// TwinCAT 3 PLC project Virtual_PLC
// ProgramVersion: 3.1.4024.0
// libraries:
//   Tc2_Standard, * (Beckhoff Automation GmbH)
//   Tc2_System, * (Beckhoff Automation GmbH)
//   Tc3_Module, * (Beckhoff Automation GmbH)
// project tree:
//   DUTs/ KlantToestand.TcDUT, KleurmachineToestand.TcDUT, MedewerkerToestand.TcDUT, schudmachineToestand.TcDUT
//   / GlobalTextList.TcGTLO, PlcTask.TcTTO, Visualization Manager.TcVMO (not stored), Visualization.TcVIS
//   GVLs/ GVL.TcGVL
//   POUs/ kleurmachine.TcPOU, Medewerker.TcPOU, Klant.TcPOU, schudmachine.TcPOU
//   VISUs/ Visu_main.TcVIS
// real-time tasks:
//   TASK PlcTask: cycle T#10ms, priority 20, ADS port 350

CONFIGURATION Virtual_PLC
    RESOURCE PLC ON TwinCAT3
        TASK PlcTask(INTERVAL := T#10ms, PRIORITY := 20);
        PROGRAM Medewerker WITH PlcTask : Medewerker;
        PROGRAM schudmachine WITH PlcTask : schudmachine;
        PROGRAM kleurmachine WITH PlcTask : kleurmachine;
        PROGRAM Klant WITH PlcTask : Klant;
    END_RESOURCE
END_CONFIGURATION

// ---- DUTs/KlantToestand.TcDUT
{attribute 'qualified_only'}
{attribute 'strict'}
TYPE KlantToestand :
(
	voorBalie := 0,
	wordtGeholpen,
	aanHetWachten,
	heeftVerf
);
END_TYPE

// ---- DUTs/KleurmachineToestand.TcDUT
{attribute 'qualified_only'}
{attribute 'strict'}
TYPE KleurmachineToestand :
(
	startup := 0,
	home,
	info,
	scan,
	wachtOpBlik,
	kleurToevoegen,
	klaarMetToevoegen
);
END_TYPE

// ---- DUTs/MedewerkerToestand.TcDUT
{attribute 'qualified_only'}
{attribute 'strict'}
TYPE MedewerkerToestand :
(
	wachtenOpKlant := 0,
	klantHelpen,
	verfMengen,
	verfGeven
);
END_TYPE

// ---- DUTs/schudmachineToestand.TcDUT
{attribute 'qualified_only'}
{attribute 'strict'}
TYPE schudmachineToestand :
(
	startup := 0,
	automode,
	blikKlemmen,
	blikSchudden
);
END_TYPE

// ---- GVLs/GVL.TcGVL
{attribute 'qualified_only'}
VAR_GLOBAL
	// Keuzes van de klant
	typeVerf 	: STRING := 'null';
	merkVerf 	: STRING := 'null';
	kleurVerf	: STRING := 'null';
	hoeveelVerf : STRING := 'null';
	
	// Opdracht voor kleurmachine
	verfOrder 	: ARRAY[1..4] OF STRING;
	
	// knoppen/sensoren kleurmachine
	homeKnop : BOOL;
	okeKnop : BOOL;
	blikPresent : BOOL;
	opdrachtKnop : BOOL;
	startKnop : BOOL;	
	
	barcodeBlik : INT;
	
	// klant variabelen
	klantWiltVerf : BOOL := TRUE;
	klantWordtGeholpen : BOOL;
	klantWacht : BOOL;
	verfAanKlantGegeven : BOOL;
	
	// schudmachine variabelen
	schudmachineReady : BOOL := FALSE;
	schudMachineBezig : BOOL := FALSE;
	deurDicht : BOOL := FALSE;
	stopSchudden : BOOL := FALSE;
END_VAR

// ---- POUs/Medewerker.TcPOU
PROGRAM Medewerker
VAR
	state : MedewerkerToestand;
	
	orderCompleet : BOOL := FALSE;
	
	medewerkerTimer : TON;
END_VAR

CASE state OF
	MedewerkerToestand.wachtenOpKlant:
		IF GVL.klantWiltVerf THEN
			state := MedewerkerToestand.klantHelpen;
		END_IF
		
	MedewerkerToestand.klantHelpen:
		// get order from customer
		GVL.klantWordtGeholpen := TRUE;
		GVL.verfOrder[1] := GVL.merkVerf;
		GVL.verfOrder[2] := GVL.kleurVerf;
		GVL.verfOrder[3] := GVL.typeVerf;
		GVL.verfOrder[4] := GVL.hoeveelVerf;
		
		IF orderCompleet THEN
			state := MedewerkerToestand.verfMengen;
		END_IF
		
	MedewerkerToestand.verfMengen:
		GVL.klantWacht := TRUE;
		medewerkerTimer(IN:= TRUE, PT:= T#7S); // Simulate the time it takes to click all buttons until scanning barcode
		// Blik onder kleurmachine zetten
		GVL.blikPresent := TRUE;
		// order aanklikken en starten
		GVL.opdrachtKnop := TRUE;
		GVL.startKnop := TRUE;
		IF medewerkerTimer.Q THEN
			// barcode scannen
		    GVL.barcodeBlik := 1234;
			GVL.opdrachtKnop := FALSE;
			GVL.startKnop := FALSE;
			IF kleurmachine.state = kleurmachineToestand.klaarMetToevoegen THEN
				GVL.blikPresent := FALSE;
				medewerkerTimer(IN:=FALSE);
				state := MedewerkerToestand.verfSchudden;
			END_IF
			
		END_IF
		
	MedewerkerToestand.verfSchudden:
		medewerkerTimer(IN:= TRUE, PT:= T#1S);
		IF NOT medewerkerTimer.Q THEN
			GVL.deurDicht := TRUE;
		ELSIF medewerkerTimer.Q AND NOT GVL.deurDicht THEN
			medewerkerTimer(IN:= FALSE);
			state := medewerkerToestand.verfGeven;
		END_IF
		
	MedewerkerToestand.verfGeven:
		GVL.klantWacht := FALSE;
		medewerkerTimer(IN:= TRUE, PT:= T#5S); // simulate giving can to customer
		IF medewerkerTimer.Q THEN
			GVL.verfAanKlantGegeven := TRUE;
			state := MedewerkerToestand.wachtenOpKlant;
			GVL.klantWordtGeholpen := FALSE;
		END_IF
		
		
END_CASE

END_PROGRAM

// ---- POUs/kleurmachine.TcPOU
PROGRAM kleurmachine
VAR
	state : KleurmachineToestand;
	
	
	kleurmachineReady : BOOL;
	kleurmachineBezig : BOOL;
	
	inputCode : INT;
	goedeCode : INT := 1234;
	
	kleurmachineTimer : TON;
END_VAR

CASE state OF
	KleurmachineToestand.startup:
		// Simulate startup
		kleurmachineTimer(IN:=TRUE, PT:=T#10S);
		IF kleurmachineTimer.Q THEN
			kleurmachineTimer(IN:=FALSE);
			state := KleurmachineToestand.home;
		END_IF
		
	KleurmachineToestand.home:
		kleurmachineReady := TRUE;
		kleurmachineBezig := FALSE;
		IF GVL.opdrachtKnop THEN
			state := KleurmachineToestand.info;
		END_IF
		
	KleurmachineToestand.info:
		IF GVL.startKnop THEN
			state := KleurmachineToestand.scan;
		END_IF
		
	KleurmachineToestand.scan:
		kleurmachineReady := FALSE;
		kleurmachineBezig := TRUE;
		IF GVL.barcodeBlik = goedeCode THEN
			state := KleurmachineToestand.wachtOpBlik;
		END_IF
		
	KleurmachineToestand.wachtOpBlik:
		IF GVL.blikPresent OR GVL.okeKnop THEN
			state := KleurmachineToestand.kleurToevoegen;
		END_IF
		
	KleurmachineToestand.kleurToevoegen:
		IF GVL.verfOrder[4] = '2.5' THEN
			kleurmachineTimer(IN:=TRUE,PT:=T#20S); // simulate the colors being added
		ELSIF GVL.verfOrder[4] = '5' THEN
			kleurmachineTimer(IN:=TRUE,PT:=T#30S); // simulate the colors being added
		ELSIF GVL.verfOrder[4] = '10' THEN
			kleurmachineTimer(IN:=TRUE,PT:=T#40S); // simulate the colors being added
		END_IF
		
		IF kleurmachineTimer.Q THEN
			state := KleurmachineToestand.klaarMetToevoegen;
		END_IF
		
	KleurmachineToestand.klaarMetToevoegen:
		IF GVL.okeKnop OR NOT GVL.blikPresent THEN
			state := KleurmachineToestand.home;	
		END_IF
END_CASE

END_PROGRAM

// ---- POUs/schudmachine.TcPOU
PROGRAM schudmachine
VAR
	State : schudmachineToestand;
	
	blikGevonden : BOOL := FALSE;
	geenBlikGevonden : BOOL;
	//fBlikKlemmen : BlikKlemmen;
	
	timerSchudMachine : TON;
	klemTimer : TON;
	blikGeklemd: BOOL;
	geenBlik: BOOL;
END_VAR

CASE State OF
	schudMachineToestand.startup:
		// Simulate startup
		timerSchudMachine(IN:=TRUE,PT:=T#5S);
		IF timerSchudMachine.Q THEN
			State := schudMachineToestand.automode;
			timerSchudMachine(IN:=FALSE);
		END_IF
		
	schudMachineToestand.automode:
		// CODE
		GVL.schudmachineReady := TRUE;
		GVL.schudmachineBezig := FALSE;
		IF GVL.deurDicht THEN
			State := schudmachineToestand.blikKlemmen;
		END_IF

	schudMachineToestand.blikKlemmen:
		// CODE
		GVL.schudmachineReady := FALSE;
		GVL.schudmachineBezig := TRUE;
		
		// clamping procedure
		klemTimer(IN:=TRUE, PT:= T#10S);
		IF klemTimer.ET = T#7S THEN // simulate finding the can with the clamp
			blikGevonden := TRUE;
			klemTimer(IN:=FALSE);
		ELSIF klemTimer.Q THEN // if no can is found
			geenBlik := TRUE;
		END_IF
		
		// checks to change state
		IF blikGevonden THEN
			State := schudmachineToestand.blikSchudden;
		ELSIF GVL.stopSchudden THEN
			State := schudmachineToestand.automode;
			GVL.deurDicht := FALSE;
		ELSIF geenBlik THEN
			State := schudmachineToestand.automode;
			GVL.deurDicht := FALSE;
		END_IF
		
	schudMachineToestand.blikSchudden:
		// CODE
		timerSchudMachine(IN:=TRUE, PT:= T#1M);
		IF timerSchudMachine.Q THEN
			State := schudmachineToestand.automode;
			GVL.deurDicht := FALSE;
		ELSIF GVL.stopSchudden THEN
			State := schudmachineToestand.automode;
			GVL.deurDicht := FALSE;
		END_IF
	
END_CASE

END_PROGRAM

// ---- POUs/Klant.TcPOU
PROGRAM Klant
VAR
	state : KlantToestand;
END_VAR

CASE state OF
	KlantToestand.voorBalie:
		IF GVL.klantWordtGeholpen THEN
			state := klantToestand.wordtGeholpen;
		END_IF
		
	KlantToestand.wordtGeholpen:
		IF GVL.klantWacht THEN
			state := KlantToestand.aanHetWachten;
		END_IF
		
	KlantToestand.aanHetWachten:
		IF GVL.verfAanKlantGegeven THEN
			state := KlantToestand.heeftVerf;
		END_IF
		
	KlantToestand.heeftVerf:
		GVL.klantWiltVerf := FALSE;
END_CASE

END_PROGRAM

// ---- GlobalTextList.TcGTLO
TEXTLIST GlobalTextList
  450 = 'Blik ja/nee'
  472 = 'Deur dicht'
  949 = 'Deur open'
  479 = 'Deur open/dicht'
  25 = 'Home'
  81 = 'Input kleur'
  893 = 'Invoer kleur'
  333 = 'Invoer liters'
  123 = 'Invoer merk'
  51 = 'Invoer verf'
  927 = 'Klant aan het wachten'
  471 = 'Klant heeft verf'
  542 = 'Klant voor balie'
  729 = 'Kleurmachine bezig'
  155 = 'Kleurmachine ready'
  838 = 'Label'
  50 = 'OK'
  138 = 'OpdrachtKnop'
  695 = 'Order compleet'
  786 = 'Schudmachine bezig'
  817 = 'Schudmachine ready'
  317 = 'Start'
  909 = 'Stop schudden'
  825 = 'Verstuur order'
  802 = 'Vul hier de gewenste kleur in'
END_TEXTLIST

// ---- Visualization.TcVIS
VISUALIZATION Visualization  // 2x2
END_VISUALIZATION

// ---- VISUs/Visu_main.TcVIS
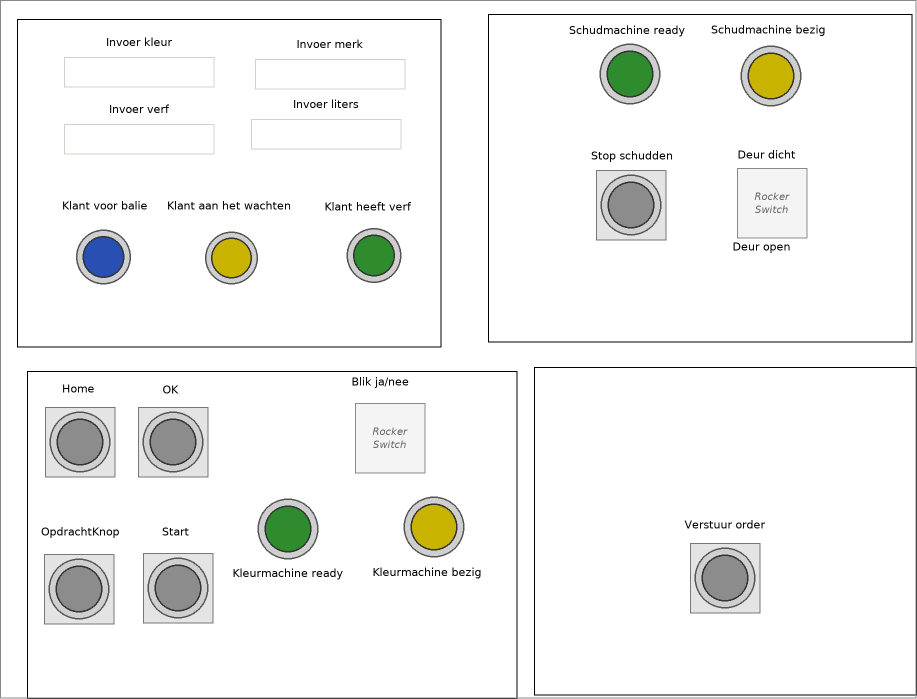
VISUALIZATION Visu_main  // 917x699
    Rectangle (534,367 383x328)
    Rectangle (488,14 424x328)
    Rectangle (17,19 424x328)
    Textfield (64,57 150x30)
        OnMouseClick: write GVL.kleurVerf via Edit
    Lamp1 (595,39 70x70), variable: GVL.schudmachineReady, style: Lamp-Lamp1-Green
    PushSwitch (596,170 70x70), variable: GVL.stopSchudden, behaviour: TAP, style: Switch-PushSwitch-Gray
    RockerSwitch (737,168 70x70), variable: GVL.deurDicht, behaviour: TOGGLE, style: Switch-RockerSwitch-Gray
    Label (716,140 101x30), "Deur dicht"
    Label (579,141 106x30), "Stop schudden"
    Label (711,232 101x30), "Deur open"
    Lamp1 (736,41 70x70), variable: GVL.schudMachineBezig, style: Lamp-Lamp1-Yellow
    Label (563,13 128x35), "Schudmachine ready"
    Label (702,15 133x30), "Schudmachine bezig"
    Label (75,25 128x35), "Invoer kleur"
    Textfield (255,59 150x30)
        OnMouseClick: write GVL.merkVerf via Edit
    Label (266,27 128x35), "Invoer merk"
    Textfield (64,124 150x30)
        OnMouseClick: write GVL.typeVerf via Edit
    Label (75,92 128x35), "Invoer verf"
    Textfield (251,119 150x30)
        OnMouseClick: write GVL.hoeveelVerf via Edit
    Label (262,87 128x35), "Invoer liters"
    PushSwitch (690,543 70x70), variable: Medewerker.orderCompleet, behaviour: TAP, style: Switch-PushSwitch-Gray
    Label (672,510 106x30), "Verstuur order"
    Rectangle (27,371 490x328)
    PushSwitch (45,407 70x70), variable: GVL.homeKnop, behaviour: TAP, style: Switch-PushSwitch-Gray
    PushSwitch (138,407 70x70), variable: GVL.okeKnop, behaviour: TAP, style: Switch-PushSwitch-Gray
    RockerSwitch (355,403 70x70), variable: GVL.blikPresent, behaviour: TOGGLE, style: Switch-RockerSwitch-Gray
    Label (39,374 79x30), "Home"
    Label (131,375 79x30), "OK"
    Label (341,367 79x30), "Blik ja/nee"
    PushSwitch (44,554 70x70), variable: GVL.opdrachtKnop, behaviour: TAP, style: Switch-PushSwitch-Gray
    PushSwitch (143,553 70x70), variable: GVL.startKnop, behaviour: TAP, style: Switch-PushSwitch-Gray
    Label (41,517 79x30), "OpdrachtKnop"
    Label (136,517 79x30), "Start"
    Lamp1 (253,494 70x70), variable: kleurmachine.kleurmachineReady, style: Lamp-Lamp1-Green
    Lamp1 (399,492 70x70), variable: kleurmachine.kleurmachineBezig, style: Lamp-Lamp1-Yellow
    Label (224,556 128x35), "Kleurmachine ready"
    Label (363,555 128x35), "Kleurmachine bezig"
    Lamp1 (201,225 61x66), variable: GVL.klantWacht, style: Lamp-Lamp1-Yellow
    Lamp1 (72,225 63x64), variable: GVL.klantWiltVerf, style: Lamp-Lamp1-Blue
    Lamp1 (337,224 74x63), variable: GVL.verfAanKlantGegeven, style: Lamp-Lamp1-Green
    Label (52,191 106x30), "Klant voor balie"
    Label (162,191 134x30), "Klant aan het wachten"
    Label (315,192 106x30), "Klant heeft verf"
END_VISUALIZATION
